{attribute 'GeneratedUsingTerminal: KL2642-0050'}
{attribute addProperty BoxType "KL2642-0050"}
{attribute addProperty Id "Channel_1AT %Q*Channel_F5DB8AD10Channel_2AT %Q*Channel_F5DB8AD10"}
{attribute addProperty CRC "4060545023"}
{attribute addProperty Size "0"}
TYPE KL_F206FFFF :
STRUCT
	{attribute addProperty Name "Channel_1"}
	Channel_1 : Channel_F5DB8AD1;
	{attribute addProperty Name "Channel_2"}
	Channel_2 : Channel_F5DB8AD1;
END_STRUCT
END_TYPE

(* stored: Version 1.2.0.0, ProductVersion 3.1.4024.9
   DUT KL_F206FFFF: Id {3f72624f-8e04-4f63-a477-e05c272efc29} *)
